FUNCTION_BLOCK Edit
VAR
	_edit : T_MaxString;
END_VAR

PROPERTY Text : STRING
GET
Text := _edit;
END_GET
SET
Text := _edit;
END_SET
END_PROPERTY

END_FUNCTION_BLOCK

(* stored: Version 1.1.0.1, ProductVersion 3.1.4024.12
   POU Edit: Id {dd182afd-7d10-410a-9d00-31674a3839a1}, SpecialFunc None
   Property Text: Id {8c53d925-f5f0-4953-a30c-774f1d18bfb3}
   Get Get: Id {1f334f1c-bb17-48ab-974e-2444e2944be4}
   Set Set: Id {ff9edd7d-ac20-4180-92ce-7533b13b0e7c} *)
